Staubli VAL3: DAEMON1.PGX

public program daemon1()
  local num l_nKey
begin

  while (getKey()!=270)
    call daemon4()
    delay(0)
  endWhile
end
